{attribute 'qualified_only'}
{attribute 'strict'}
{attribute 'to_string'}
TYPE StackerCraneSteps :
(
	Waiting := 0,
	DriveToLoadingPosition,
	ForkUnderLoad,
	LiftLoadItem,
	ForkToMiddle,
	DriveToUnloadPrePosition,
	ForkInWarehouse,
	DriveToUnloadPosition
);
END_TYPE

(* stored: Version 1.1.0.1
   DUT StackerCraneSteps: Id {ad15095a-c874-4d94-aa8b-9e325c07147b} *)
